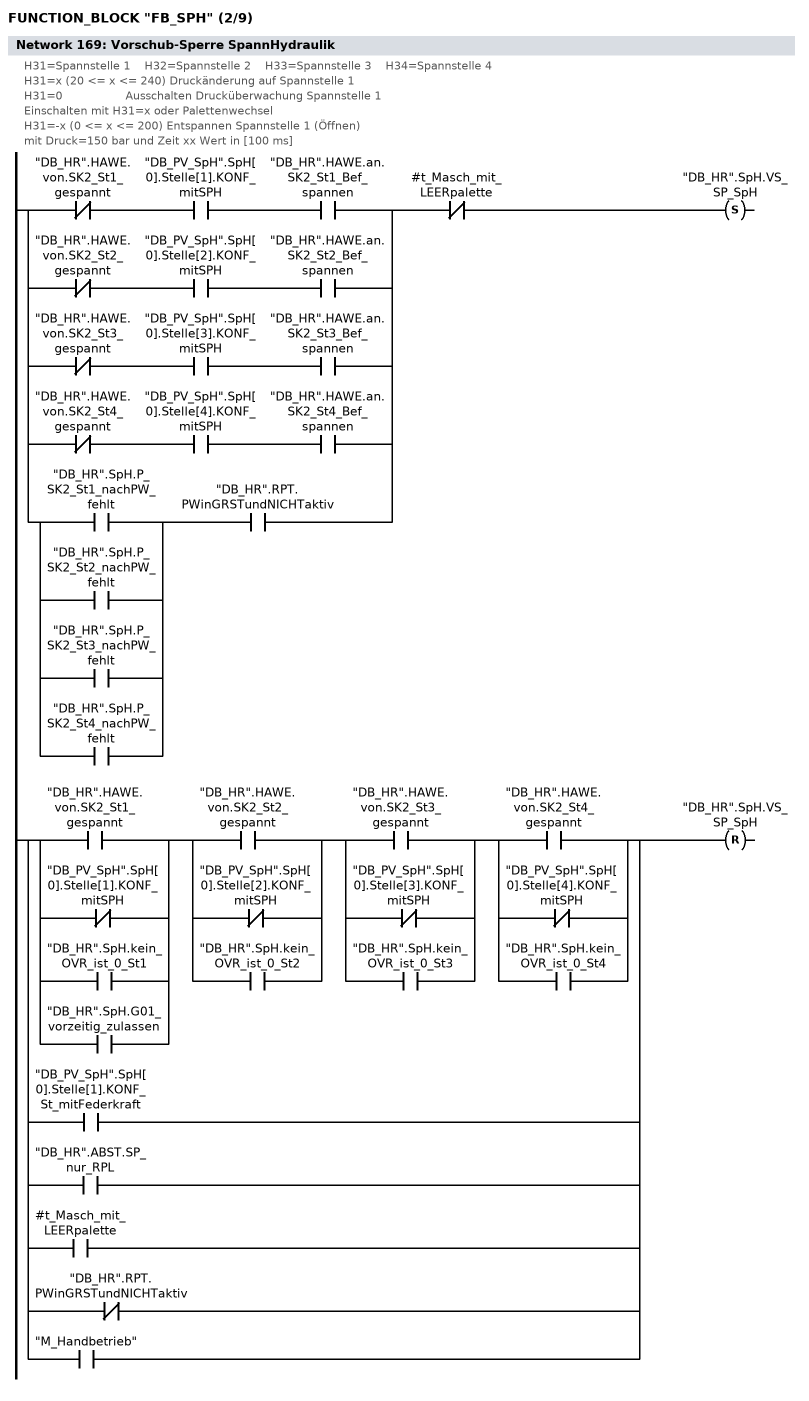
      U(    ;
      UN    "DB_HR".HAWE.von.SK2_St1_gespannt;
      U     "DB_PV_SpH".SpH[0].Stelle[1].KONF_mitSPH;
      U     "DB_HR".HAWE.an.SK2_St1_Bef_spannen;
      O     ;
      UN    "DB_HR".HAWE.von.SK2_St2_gespannt;
      U     "DB_PV_SpH".SpH[0].Stelle[2].KONF_mitSPH;
      U     "DB_HR".HAWE.an.SK2_St2_Bef_spannen;
      O     ;
      UN    "DB_HR".HAWE.von.SK2_St3_gespannt;
      U     "DB_PV_SpH".SpH[0].Stelle[3].KONF_mitSPH;
      U     "DB_HR".HAWE.an.SK2_St3_Bef_spannen;
      O     ;
      UN    "DB_HR".HAWE.von.SK2_St4_gespannt;
      U     "DB_PV_SpH".SpH[0].Stelle[4].KONF_mitSPH;
      U     "DB_HR".HAWE.an.SK2_St4_Bef_spannen;
      O     ;
      U(    ;
      O     "DB_HR".SpH.P_SK2_St1_nachPW_fehlt;
      O     "DB_HR".SpH.P_SK2_St2_nachPW_fehlt;
      O     "DB_HR".SpH.P_SK2_St3_nachPW_fehlt;
      O     "DB_HR".SpH.P_SK2_St4_nachPW_fehlt;
      )     ;
      U     "DB_HR".RPT.PWinGRSTundNICHTaktiv;
      )     ;
      UN    #t_Masch_mit_LEERpalette;

      S     "DB_HR".SpH.VS_SP_SpH;
      U(    ;
      U(    ;
      O     "DB_HR".HAWE.von.SK2_St1_gespannt;
      ON    "DB_PV_SpH".SpH[0].Stelle[1].KONF_mitSPH;
      O     "DB_HR".SpH.kein_OVR_ist_0_St1;
      O     "DB_HR".SpH.G01_vorzeitig_zulassen;
      )     ;
      U(    ;
      O     "DB_HR".HAWE.von.SK2_St2_gespannt;
      ON    "DB_PV_SpH".SpH[0].Stelle[2].KONF_mitSPH;
      O     "DB_HR".SpH.kein_OVR_ist_0_St2;
      )     ;
      U(    ;
      O     "DB_HR".HAWE.von.SK2_St3_gespannt;
      ON    "DB_PV_SpH".SpH[0].Stelle[3].KONF_mitSPH;
      O     "DB_HR".SpH.kein_OVR_ist_0_St3;
      )     ;
      U(    ;
      O     "DB_HR".HAWE.von.SK2_St4_gespannt;
      ON    "DB_PV_SpH".SpH[0].Stelle[4].KONF_mitSPH;
      O     "DB_HR".SpH.kein_OVR_ist_0_St4;
      )     ;
      O     "DB_PV_SpH".SpH[0].Stelle[1].KONF_St_mitFederkraft;
      O     "DB_HR".ABST.SP_nur_RPL;
      O     #t_Masch_mit_LEERpalette;
      ON    "DB_HR".RPT.PWinGRSTundNICHTaktiv;
      O     "M_Handbetrieb";
      )     ;
      R     "DB_HR".SpH.VS_SP_SpH;
      NOP   0;
NETWORK
TITLE =700451 VS-SP SpannHydraulik nicht hochgefahren
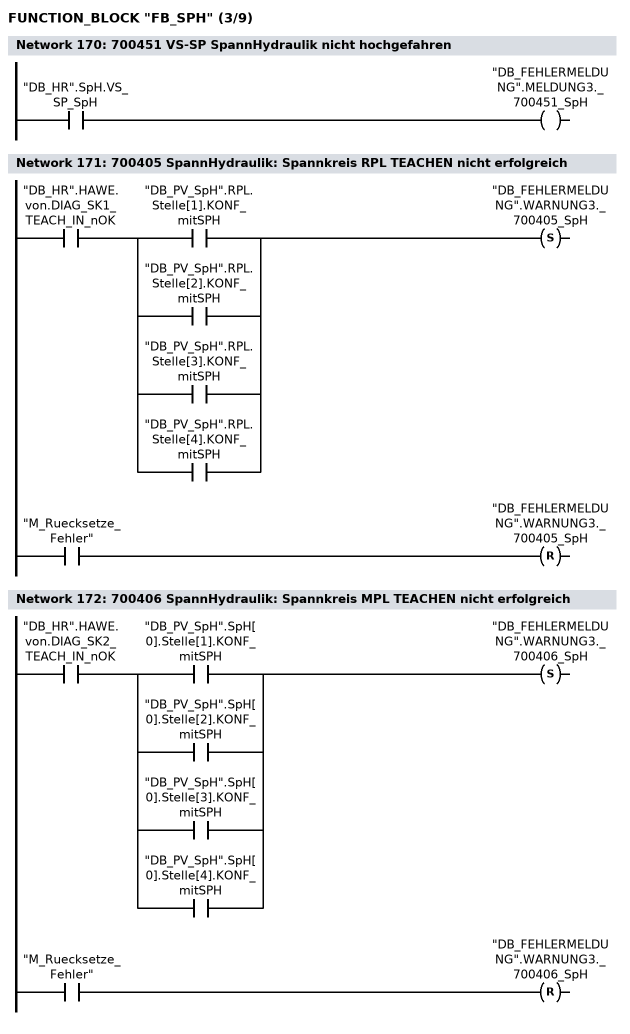

      U     "DB_HR".SpH.VS_SP_SpH;
      =     "DB_FEHLERMELDUNG".MELDUNG3._700451_SpH;
NETWORK
TITLE =700405 SpannHydraulik: Spannkreis RPL TEACHEN nicht erfolgreich

      U     "DB_HR".HAWE.von.DIAG_SK1_TEACH_IN_nOK;
      U(    ;
      O     "DB_PV_SpH".RPL.Stelle[1].KONF_mitSPH;
      O     "DB_PV_SpH".RPL.Stelle[2].KONF_mitSPH;
      O     "DB_PV_SpH".RPL.Stelle[3].KONF_mitSPH;
      O     "DB_PV_SpH".RPL.Stelle[4].KONF_mitSPH;
      )     ;
      S     "DB_FEHLERMELDUNG".WARNUNG3._700405_SpH;
      U     "M_Ruecksetze_Fehler";
      R     "DB_FEHLERMELDUNG".WARNUNG3._700405_SpH;
      NOP   0;
NETWORK
TITLE =700406 SpannHydraulik: Spannkreis MPL TEACHEN nicht erfolgreich

      U     "DB_HR".HAWE.von.DIAG_SK2_TEACH_IN_nOK;
      U(    ;
      O     "DB_PV_SpH".SpH[0].Stelle[1].KONF_mitSPH;
      O     "DB_PV_SpH".SpH[0].Stelle[2].KONF_mitSPH;
      O     "DB_PV_SpH".SpH[0].Stelle[3].KONF_mitSPH;
      O     "DB_PV_SpH".SpH[0].Stelle[4].KONF_mitSPH;
      )     ;
      S     "DB_FEHLERMELDUNG".WARNUNG3._700406_SpH;
      U     "M_Ruecksetze_Fehler";
      R     "DB_FEHLERMELDUNG".WARNUNG3._700406_SpH;
      NOP   0;
NETWORK
TITLE =700414 von HAWEbox: Spannkreis RPL Druck nicht erreichbar
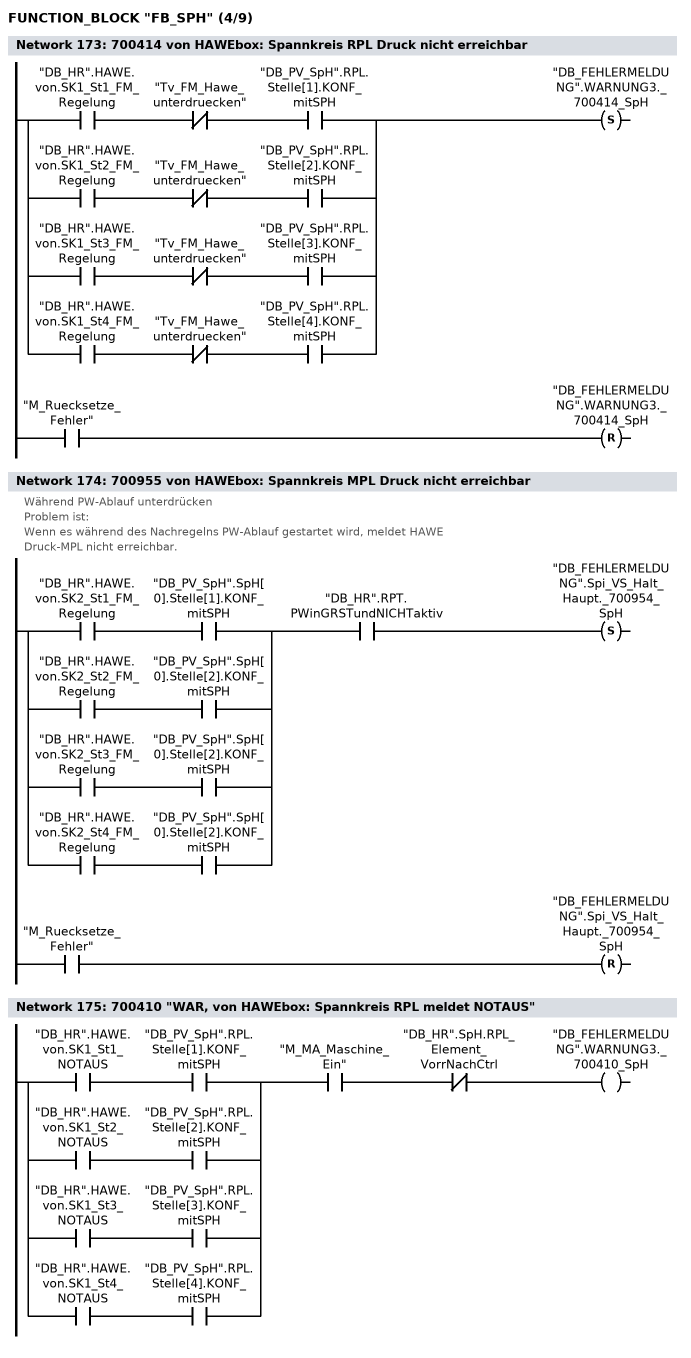

      U(    ;
      U     "DB_HR".HAWE.von.SK1_St1_FM_Regelung;
      UN    "Tv_FM_Hawe_unterdruecken";
      U     "DB_PV_SpH".RPL.Stelle[1].KONF_mitSPH;
      O     ;
      U     "DB_HR".HAWE.von.SK1_St2_FM_Regelung;
      UN    "Tv_FM_Hawe_unterdruecken";
      U     "DB_PV_SpH".RPL.Stelle[2].KONF_mitSPH;
      O     ;
      U     "DB_HR".HAWE.von.SK1_St3_FM_Regelung;
      UN    "Tv_FM_Hawe_unterdruecken";
      U     "DB_PV_SpH".RPL.Stelle[3].KONF_mitSPH;
      O     ;
      U     "DB_HR".HAWE.von.SK1_St4_FM_Regelung;
      UN    "Tv_FM_Hawe_unterdruecken";
      U     "DB_PV_SpH".RPL.Stelle[4].KONF_mitSPH;
      )     ;
      S     "DB_FEHLERMELDUNG".WARNUNG3._700414_SpH;

      U     "M_Ruecksetze_Fehler";
      R     "DB_FEHLERMELDUNG".WARNUNG3._700414_SpH;
      NOP   0;
NETWORK
TITLE =700955 von HAWEbox: Spannkreis MPL Druck nicht erreichbar
//Während PW-Ablauf unterdrücken
//Problem ist:
//Wenn es während des Nachregelns PW-Ablauf gestartet wird, meldet HAWE
//Druck-MPL nicht erreichbar.
      U(    ;
      U     "DB_HR".HAWE.von.SK2_St1_FM_Regelung;
      U     "DB_PV_SpH".SpH[0].Stelle[1].KONF_mitSPH;
      O     ;
      U     "DB_HR".HAWE.von.SK2_St2_FM_Regelung;
      U     "DB_PV_SpH".SpH[0].Stelle[2].KONF_mitSPH;
      O     ;
      U     "DB_HR".HAWE.von.SK2_St3_FM_Regelung;
      U     "DB_PV_SpH".SpH[0].Stelle[2].KONF_mitSPH;
      O     ;
      U     "DB_HR".HAWE.von.SK2_St4_FM_Regelung;
      U     "DB_PV_SpH".SpH[0].Stelle[2].KONF_mitSPH;
      )     ;
      U     "DB_HR".RPT.PWinGRSTundNICHTaktiv;

      S     "DB_FEHLERMELDUNG".Spi_VS_Halt_Haupt._700954_SpH;
      U     "M_Ruecksetze_Fehler";
      R     "DB_FEHLERMELDUNG".Spi_VS_Halt_Haupt._700954_SpH;
      NOP   0;
NETWORK
TITLE =700410 "WAR, von HAWEbox: Spannkreis RPL meldet NOTAUS"

      U(    ;
      U     "DB_HR".HAWE.von.SK1_St1_NOTAUS;
      U     "DB_PV_SpH".RPL.Stelle[1].KONF_mitSPH;
      O     ;
      U     "DB_HR".HAWE.von.SK1_St2_NOTAUS;
      U     "DB_PV_SpH".RPL.Stelle[2].KONF_mitSPH;
      O     ;
      U     "DB_HR".HAWE.von.SK1_St3_NOTAUS;
      U     "DB_PV_SpH".RPL.Stelle[3].KONF_mitSPH;
      O     ;
      U     "DB_HR".HAWE.von.SK1_St4_NOTAUS;
      U     "DB_PV_SpH".RPL.Stelle[4].KONF_mitSPH;
      )     ;
      U     "M_MA_Maschine_Ein";
      UN    "DB_HR".SpH.RPL_Element_VorrNachCtrl;
      =     "DB_FEHLERMELDUNG".WARNUNG3._700410_SpH;
NETWORK
TITLE =700411 "WAR, von HAWEbox: Spannkreis MPL meldet NOTAUS"
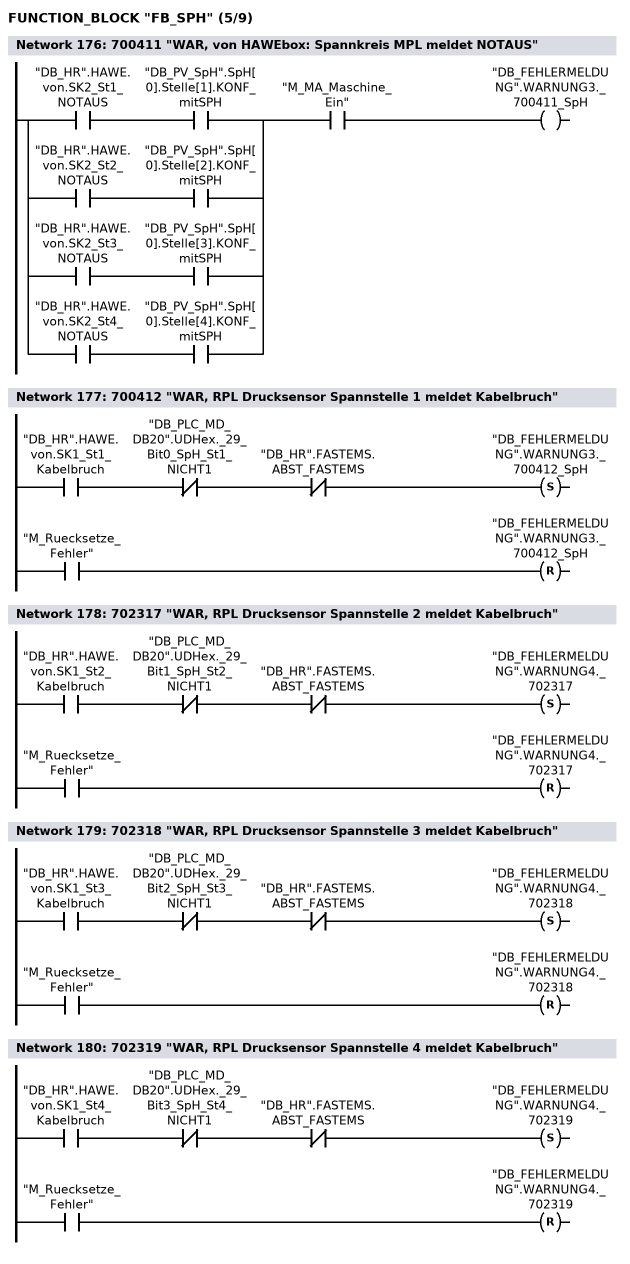

      U(    ;
      U     "DB_HR".HAWE.von.SK2_St1_NOTAUS;
      U     "DB_PV_SpH".SpH[0].Stelle[1].KONF_mitSPH;
      O     ;
      U     "DB_HR".HAWE.von.SK2_St2_NOTAUS;
      U     "DB_PV_SpH".SpH[0].Stelle[2].KONF_mitSPH;
      O     ;
      U     "DB_HR".HAWE.von.SK2_St3_NOTAUS;
      U     "DB_PV_SpH".SpH[0].Stelle[3].KONF_mitSPH;
      O     ;
      U     "DB_HR".HAWE.von.SK2_St4_NOTAUS;
      U     "DB_PV_SpH".SpH[0].Stelle[4].KONF_mitSPH;
      )     ;
      U     "M_MA_Maschine_Ein";
      =     "DB_FEHLERMELDUNG".WARNUNG3._700411_SpH;
NETWORK
TITLE =700412 "WAR, RPL Drucksensor Spannstelle 1 meldet Kabelbruch"

      U     "DB_HR".HAWE.von.SK1_St1_Kabelbruch;
      UN    "DB_PLC_MD_DB20".UDHex._29_Bit0_SpH_St1_NICHT1;
      UN    "DB_HR".FASTEMS.ABST_FASTEMS;
      S     "DB_FEHLERMELDUNG".WARNUNG3._700412_SpH;
      U     "M_Ruecksetze_Fehler";
      R     "DB_FEHLERMELDUNG".WARNUNG3._700412_SpH;
      NOP   0;
NETWORK
TITLE =702317 "WAR, RPL Drucksensor Spannstelle 2 meldet Kabelbruch"

      U     "DB_HR".HAWE.von.SK1_St2_Kabelbruch;
      UN    "DB_PLC_MD_DB20".UDHex._29_Bit1_SpH_St2_NICHT1;
      UN    "DB_HR".FASTEMS.ABST_FASTEMS;
      S     "DB_FEHLERMELDUNG".WARNUNG4._702317;
      U     "M_Ruecksetze_Fehler";
      R     "DB_FEHLERMELDUNG".WARNUNG4._702317;
      NOP   0;
NETWORK
TITLE =702318 "WAR, RPL Drucksensor Spannstelle 3 meldet Kabelbruch"

      U     "DB_HR".HAWE.von.SK1_St3_Kabelbruch;
      UN    "DB_PLC_MD_DB20".UDHex._29_Bit2_SpH_St3_NICHT1;
      UN    "DB_HR".FASTEMS.ABST_FASTEMS;
      S     "DB_FEHLERMELDUNG".WARNUNG4._702318;
      U     "M_Ruecksetze_Fehler";
      R     "DB_FEHLERMELDUNG".WARNUNG4._702318;
      NOP   0;
NETWORK
TITLE =702319 "WAR, RPL Drucksensor Spannstelle 4 meldet Kabelbruch"

      U     "DB_HR".HAWE.von.SK1_St4_Kabelbruch;
      UN    "DB_PLC_MD_DB20".UDHex._29_Bit3_SpH_St4_NICHT1;
      UN    "DB_HR".FASTEMS.ABST_FASTEMS;
      S     "DB_FEHLERMELDUNG".WARNUNG4._702319;
      U     "M_Ruecksetze_Fehler";
      R     "DB_FEHLERMELDUNG".WARNUNG4._702319;
      NOP   0;
NETWORK
TITLE =FM: RPL PROP-Ventil Kabelbruch
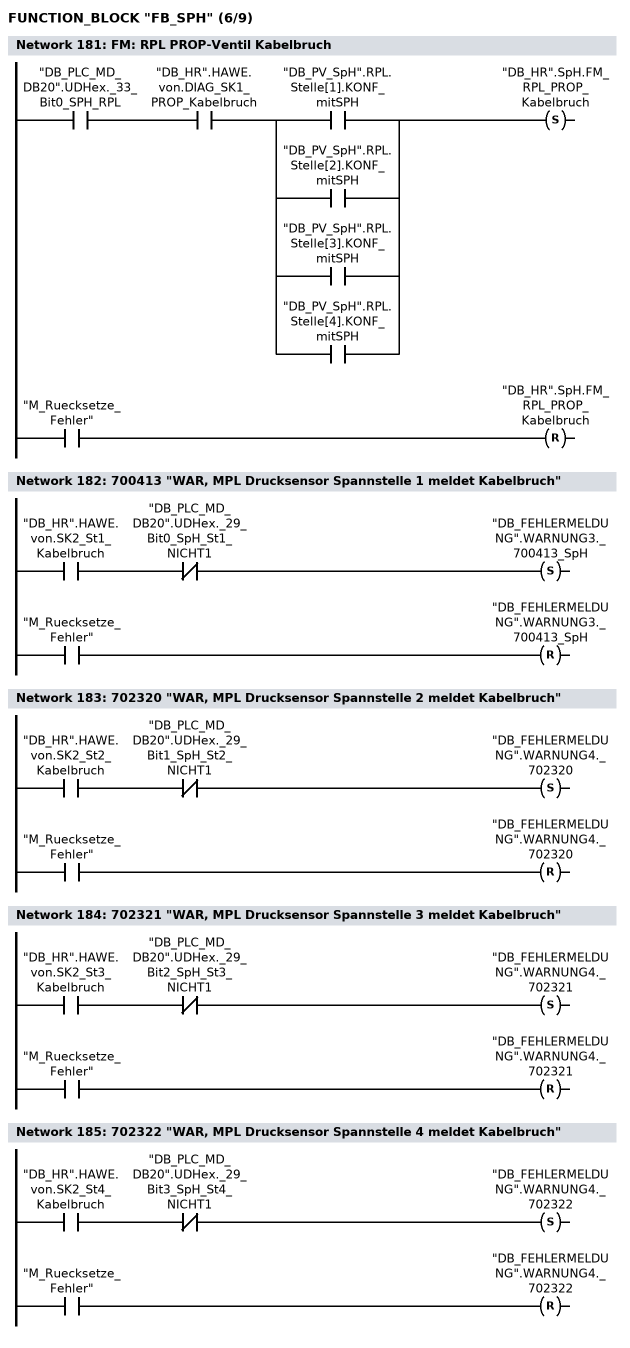

      U     "DB_PLC_MD_DB20".UDHex._33_Bit0_SPH_RPL;
      U     "DB_HR".HAWE.von.DIAG_SK1_PROP_Kabelbruch;
      U(    ;
      O     "DB_PV_SpH".RPL.Stelle[1].KONF_mitSPH;
      O     "DB_PV_SpH".RPL.Stelle[2].KONF_mitSPH;
      O     "DB_PV_SpH".RPL.Stelle[3].KONF_mitSPH;
      O     "DB_PV_SpH".RPL.Stelle[4].KONF_mitSPH;
      )     ;
      S     "DB_HR".SpH.FM_RPL_PROP_Kabelbruch;
      U     "M_Ruecksetze_Fehler";
      R     "DB_HR".SpH.FM_RPL_PROP_Kabelbruch;
      NOP   0;
NETWORK
TITLE =700413 "WAR, MPL Drucksensor Spannstelle 1 meldet Kabelbruch"

      U     "DB_HR".HAWE.von.SK2_St1_Kabelbruch;
      UN    "DB_PLC_MD_DB20".UDHex._29_Bit0_SpH_St1_NICHT1;
      S     "DB_FEHLERMELDUNG".WARNUNG3._700413_SpH;
      U     "M_Ruecksetze_Fehler";
      R     "DB_FEHLERMELDUNG".WARNUNG3._700413_SpH;
      NOP   0;
NETWORK
TITLE =702320 "WAR, MPL Drucksensor Spannstelle 2 meldet Kabelbruch"

      U     "DB_HR".HAWE.von.SK2_St2_Kabelbruch;
      UN    "DB_PLC_MD_DB20".UDHex._29_Bit1_SpH_St2_NICHT1;
      S     "DB_FEHLERMELDUNG".WARNUNG4._702320;
      U     "M_Ruecksetze_Fehler";
      R     "DB_FEHLERMELDUNG".WARNUNG4._702320;
      NOP   0;
NETWORK
TITLE =702321 "WAR, MPL Drucksensor Spannstelle 3 meldet Kabelbruch"

      U     "DB_HR".HAWE.von.SK2_St3_Kabelbruch;
      UN    "DB_PLC_MD_DB20".UDHex._29_Bit2_SpH_St3_NICHT1;
      S     "DB_FEHLERMELDUNG".WARNUNG4._702321;
      U     "M_Ruecksetze_Fehler";
      R     "DB_FEHLERMELDUNG".WARNUNG4._702321;
      NOP   0;
NETWORK
TITLE =702322 "WAR, MPL Drucksensor Spannstelle 4 meldet Kabelbruch"

      U     "DB_HR".HAWE.von.SK2_St4_Kabelbruch;
      UN    "DB_PLC_MD_DB20".UDHex._29_Bit3_SpH_St4_NICHT1;
      S     "DB_FEHLERMELDUNG".WARNUNG4._702322;
      U     "M_Ruecksetze_Fehler";
      R     "DB_FEHLERMELDUNG".WARNUNG4._702322;
      NOP   0;
NETWORK
TITLE =FM: MPL PROP-Ventil Kabelbruch
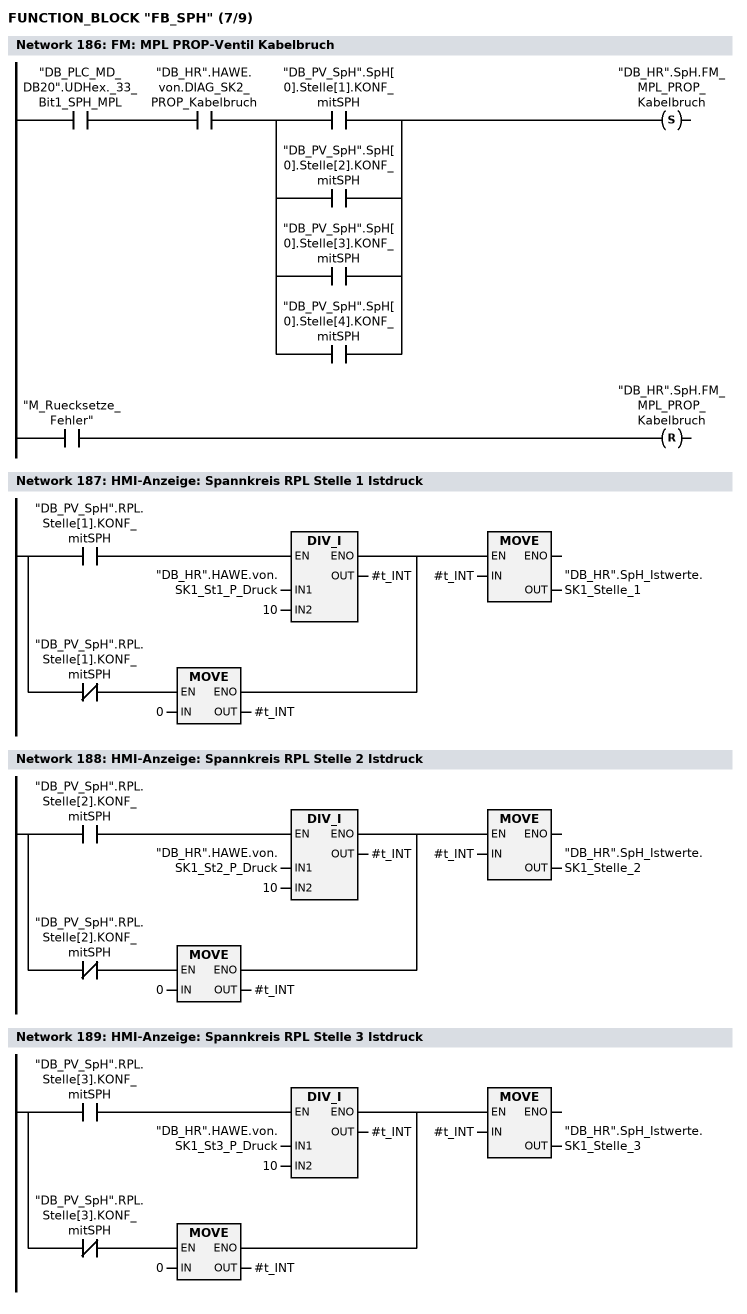

      U     "DB_PLC_MD_DB20".UDHex._33_Bit1_SPH_MPL;
      U     "DB_HR".HAWE.von.DIAG_SK2_PROP_Kabelbruch;
      U(    ;
      O     "DB_PV_SpH".SpH[0].Stelle[1].KONF_mitSPH;
      O     "DB_PV_SpH".SpH[0].Stelle[2].KONF_mitSPH;
      O     "DB_PV_SpH".SpH[0].Stelle[3].KONF_mitSPH;
      O     "DB_PV_SpH".SpH[0].Stelle[4].KONF_mitSPH;
      )     ;
      S     "DB_HR".SpH.FM_MPL_PROP_Kabelbruch;
      U     "M_Ruecksetze_Fehler";
      R     "DB_HR".SpH.FM_MPL_PROP_Kabelbruch;
      NOP   0;
NETWORK
TITLE =HMI-Anzeige: Spannkreis RPL Stelle 1 Istdruck

      U(    ;
      O(    ;
      U     "DB_PV_SpH".RPL.Stelle[1].KONF_mitSPH;
      SPBNB _01b;
      L     "DB_HR".HAWE.von.SK1_St1_P_Druck;
      L     10;
      /I    ;
      T     #t_INT;
      UN    OV;
      SAVE  ;
      CLR   ;
_01b: U     BIE;
      )     ;
      O(    ;
      UN    "DB_PV_SpH".RPL.Stelle[1].KONF_mitSPH;
      SPBNB _028;
      L     0;
      T     #t_INT;
      SET   ;
      SAVE  ;
      CLR   ;
_028: U     BIE;
      )     ;
      )     ;
      SPBNB _029;
      L     #t_INT;
      T     "DB_HR".SpH_Istwerte.SK1_Stelle_1;
_029: NOP   0;
NETWORK
TITLE =HMI-Anzeige: Spannkreis RPL Stelle 2 Istdruck

      U(    ;
      O(    ;
      U     "DB_PV_SpH".RPL.Stelle[2].KONF_mitSPH;
      SPBNB _02a;
      L     "DB_HR".HAWE.von.SK1_St2_P_Druck;
      L     10;
      /I    ;
      T     #t_INT;
      UN    OV;
      SAVE  ;
      CLR   ;
_02a: U     BIE;
      )     ;
      O(    ;
      UN    "DB_PV_SpH".RPL.Stelle[2].KONF_mitSPH;
      SPBNB _02b;
      L     0;
      T     #t_INT;
      SET   ;
      SAVE  ;
      CLR   ;
_02b: U     BIE;
      )     ;
      )     ;
      SPBNB _02f;
      L     #t_INT;
      T     "DB_HR".SpH_Istwerte.SK1_Stelle_2;
_02f: NOP   0;
NETWORK
TITLE =HMI-Anzeige: Spannkreis RPL Stelle 3 Istdruck

      U(    ;
      O(    ;
      U     "DB_PV_SpH".RPL.Stelle[3].KONF_mitSPH;
      SPBNB _034;
      L     "DB_HR".HAWE.von.SK1_St3_P_Druck;
      L     10;
      /I    ;
      T     #t_INT;
      UN    OV;
      SAVE  ;
      CLR   ;
_034: U     BIE;
      )     ;
      O(    ;
      UN    "DB_PV_SpH".RPL.Stelle[3].KONF_mitSPH;
      SPBNB _035;
      L     0;
      T     #t_INT;
      SET   ;
      SAVE  ;
      CLR   ;
_035: U     BIE;
      )     ;
      )     ;
      SPBNB _036;
      L     #t_INT;
      T     "DB_HR".SpH_Istwerte.SK1_Stelle_3;
_036: NOP   0;
NETWORK
TITLE =HMI-Anzeige: Spannkreis RPL Stelle 4 Istdruck
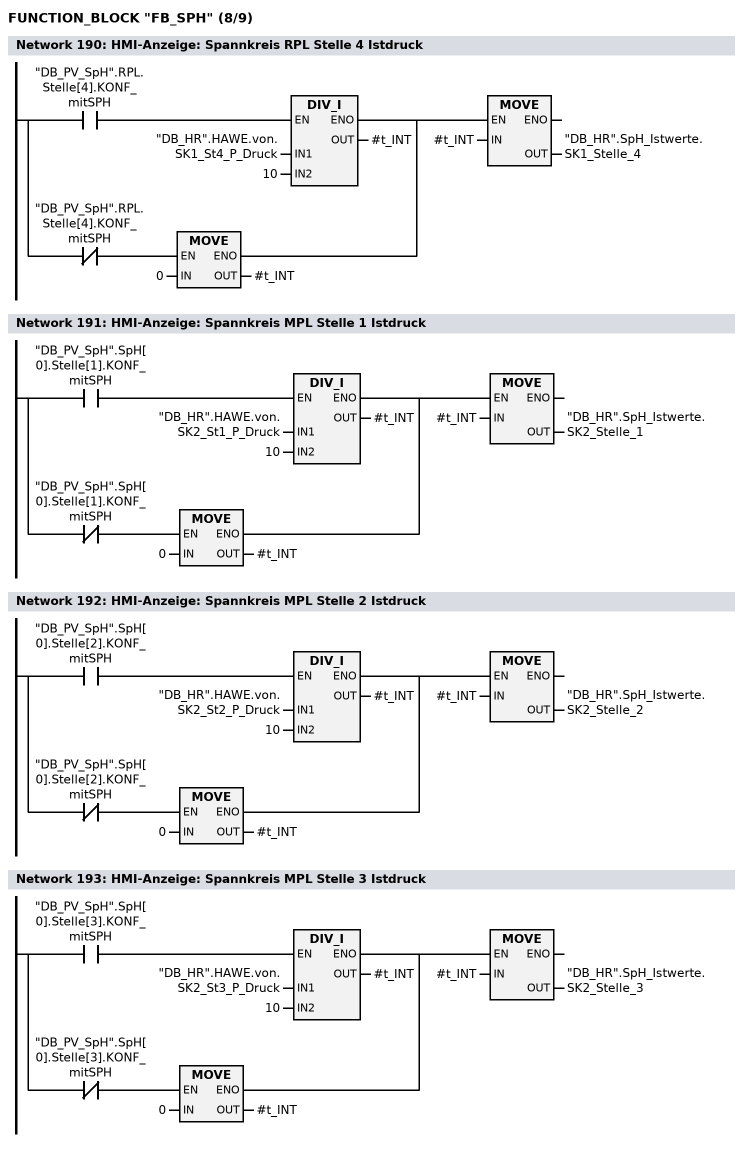

      U(    ;
      O(    ;
      U     "DB_PV_SpH".RPL.Stelle[4].KONF_mitSPH;
      SPBNB _037;
      L     "DB_HR".HAWE.von.SK1_St4_P_Druck;
      L     10;
      /I    ;
      T     #t_INT;
      UN    OV;
      SAVE  ;
      CLR   ;
_037: U     BIE;
      )     ;
      O(    ;
      UN    "DB_PV_SpH".RPL.Stelle[4].KONF_mitSPH;
      SPBNB _038;
      L     0;
      T     #t_INT;
      SET   ;
      SAVE  ;
      CLR   ;
_038: U     BIE;
      )     ;
      )     ;
      SPBNB _039;
      L     #t_INT;
      T     "DB_HR".SpH_Istwerte.SK1_Stelle_4;
_039: NOP   0;
NETWORK
TITLE =HMI-Anzeige: Spannkreis MPL Stelle 1 Istdruck

      U(    ;
      O(    ;
      U     "DB_PV_SpH".SpH[0].Stelle[1].KONF_mitSPH;
      SPBNB _03a;
      L     "DB_HR".HAWE.von.SK2_St1_P_Druck;
      L     10;
      /I    ;
      T     #t_INT;
      UN    OV;
      SAVE  ;
      CLR   ;
_03a: U     BIE;
      )     ;
      O(    ;
      UN    "DB_PV_SpH".SpH[0].Stelle[1].KONF_mitSPH;
      SPBNB _03b;
      L     0;
      T     #t_INT;
      SET   ;
      SAVE  ;
      CLR   ;
_03b: U     BIE;
      )     ;
      )     ;
      SPBNB _03f;
      L     #t_INT;
      T     "DB_HR".SpH_Istwerte.SK2_Stelle_1;
_03f: NOP   0;
NETWORK
TITLE =HMI-Anzeige: Spannkreis MPL Stelle 2 Istdruck

      U(    ;
      O(    ;
      U     "DB_PV_SpH".SpH[0].Stelle[2].KONF_mitSPH;
      SPBNB _04c;
      L     "DB_HR".HAWE.von.SK2_St2_P_Druck;
      L     10;
      /I    ;
      T     #t_INT;
      UN    OV;
      SAVE  ;
      CLR   ;
_04c: U     BIE;
      )     ;
      O(    ;
      UN    "DB_PV_SpH".SpH[0].Stelle[2].KONF_mitSPH;
      SPBNB _04d;
      L     0;
      T     #t_INT;
      SET   ;
      SAVE  ;
      CLR   ;
_04d: U     BIE;
      )     ;
      )     ;
      SPBNB _04e;
      L     #t_INT;
      T     "DB_HR".SpH_Istwerte.SK2_Stelle_2;
_04e: NOP   0;
NETWORK
TITLE =HMI-Anzeige: Spannkreis MPL Stelle 3 Istdruck

      U(    ;
      O(    ;
      U     "DB_PV_SpH".SpH[0].Stelle[3].KONF_mitSPH;
      SPBNB _04f;
      L     "DB_HR".HAWE.von.SK2_St3_P_Druck;
      L     10;
      /I    ;
      T     #t_INT;
      UN    OV;
      SAVE  ;
      CLR   ;
_04f: U     BIE;
      )     ;
      O(    ;
      UN    "DB_PV_SpH".SpH[0].Stelle[3].KONF_mitSPH;
      SPBNB _053;
      L     0;
      T     #t_INT;
      SET   ;
      SAVE  ;
      CLR   ;
_053: U     BIE;
      )     ;
      )     ;
      SPBNB _058;
      L     #t_INT;
      T     "DB_HR".SpH_Istwerte.SK2_Stelle_3;
_058: NOP   0;
NETWORK
TITLE =HMI-Anzeige: Spannkreis MPL Stelle 4 Istdruck
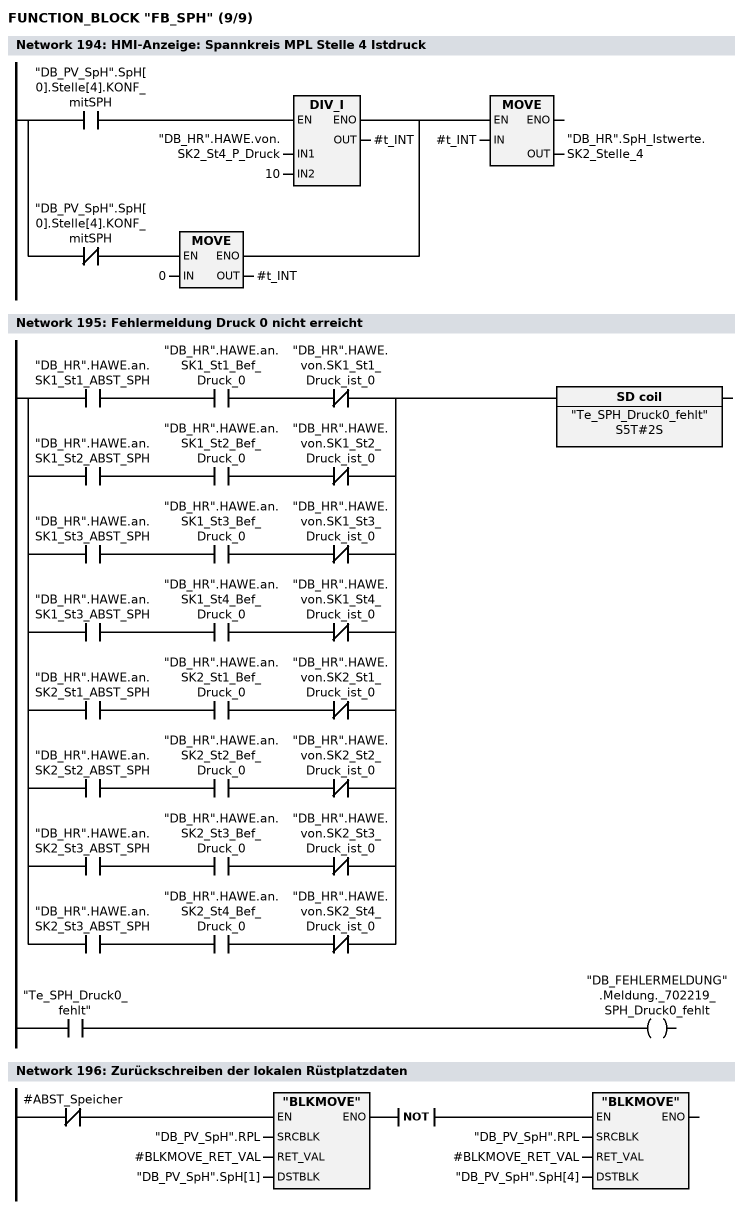

      U(    ;
      O(    ;
      U     "DB_PV_SpH".SpH[0].Stelle[4].KONF_mitSPH;
      SPBNB _059;
      L     "DB_HR".HAWE.von.SK2_St4_P_Druck;
      L     10;
      /I    ;
      T     #t_INT;
      UN    OV;
      SAVE  ;
      CLR   ;
_059: U     BIE;
      )     ;
      O(    ;
      UN    "DB_PV_SpH".SpH[0].Stelle[4].KONF_mitSPH;
      SPBNB _05a;
      L     0;
      T     #t_INT;
      SET   ;
      SAVE  ;
      CLR   ;
_05a: U     BIE;
      )     ;
      )     ;
      SPBNB _05b;
      L     #t_INT;
      T     "DB_HR".SpH_Istwerte.SK2_Stelle_4;
_05b: NOP   0;
NETWORK
TITLE =Fehlermeldung Druck 0 nicht erreicht

      U(    ;
      U     "DB_HR".HAWE.an.SK1_St1_ABST_SPH;
      U     "DB_HR".HAWE.an.SK1_St1_Bef_Druck_0;
      UN    "DB_HR".HAWE.von.SK1_St1_Druck_ist_0;
      O     ;
      U     "DB_HR".HAWE.an.SK1_St2_ABST_SPH;
      U     "DB_HR".HAWE.an.SK1_St2_Bef_Druck_0;
      UN    "DB_HR".HAWE.von.SK1_St2_Druck_ist_0;
      O     ;
      U     "DB_HR".HAWE.an.SK1_St3_ABST_SPH;
      U     "DB_HR".HAWE.an.SK1_St3_Bef_Druck_0;
      UN    "DB_HR".HAWE.von.SK1_St3_Druck_ist_0;
      O     ;
      U     "DB_HR".HAWE.an.SK1_St3_ABST_SPH;
      U     "DB_HR".HAWE.an.SK1_St4_Bef_Druck_0;
      UN    "DB_HR".HAWE.von.SK1_St4_Druck_ist_0;
      O     ;
      U     "DB_HR".HAWE.an.SK2_St1_ABST_SPH;
      U     "DB_HR".HAWE.an.SK2_St1_Bef_Druck_0;
      UN    "DB_HR".HAWE.von.SK2_St1_Druck_ist_0;
      O     ;
      U     "DB_HR".HAWE.an.SK2_St2_ABST_SPH;
      U     "DB_HR".HAWE.an.SK2_St2_Bef_Druck_0;
      UN    "DB_HR".HAWE.von.SK2_St2_Druck_ist_0;
      O     ;
      U     "DB_HR".HAWE.an.SK2_St3_ABST_SPH;
      U     "DB_HR".HAWE.an.SK2_St3_Bef_Druck_0;
      UN    "DB_HR".HAWE.von.SK2_St3_Druck_ist_0;
      O     ;
      U     "DB_HR".HAWE.an.SK2_St3_ABST_SPH;
      U     "DB_HR".HAWE.an.SK2_St4_Bef_Druck_0;
      UN    "DB_HR".HAWE.von.SK2_St4_Druck_ist_0;
      )     ;
      L     S5T#2S;
      SE    "Te_SPH_Druck0_fehlt";
      NOP   0;
      NOP   0;
      NOP   0;
      U     "Te_SPH_Druck0_fehlt";
      =     "DB_FEHLERMELDUNG".Meldung._702219_SPH_Druck0_fehlt;
NETWORK
TITLE =Zurückschreiben der lokalen Rüstplatzdaten

      U(    ;
      UN    #ABST_Speicher;
      SPBNB _05c;
      CALL "BLKMOVE" (
           SRCBLK                   := "DB_PV_SpH".RPL,
           RET_VAL                  := #BLKMOVE_RET_VAL,
           DSTBLK                   := "DB_PV_SpH".SpH[1]);
_05c: U     BIE;
      )     ;
      NOT   ;
      SPBNB _05d;
      CALL "BLKMOVE" (
           SRCBLK                   := "DB_PV_SpH".RPL,
           RET_VAL                  := #BLKMOVE_RET_VAL,
           DSTBLK                   := "DB_PV_SpH".SpH[4]);
_05d: NOP   0;
END_FUNCTION_BLOCK

